// TIA Portal V20 export
DATA_BLOCK "DB_Components"   // DB119
// stored: InstanceOfName FB_Components, InstanceOfType FB
"FB_Components"
   // VAR
   //    sRT_Update : R_TRIG;
   //    sShuttle1DrilledPart : "FB_OPC_PartStatus";
   //    sShuttle1UndrilledPart { S7_SetPoint := 'True'} : "FB_OPC_PartStatus";
   //    sShuttle2DrilledPart { S7_SetPoint := 'True'} : "FB_OPC_PartStatus";
   //    sShuttle2UndrilledPart { S7_SetPoint := 'True'} : "FB_OPC_PartStatus";
   //    sShuttle1DrilledBw : "FB_OPC_PartStatus";
   //    sShuttle1UndrilledBw { S7_SetPoint := 'True'} : "FB_OPC_PartStatus";
   //    sShuttle2DrilledBw { S7_SetPoint := 'True'} : "FB_OPC_PartStatus";
   //    sShuttle2UndrilledBw { S7_SetPoint := 'True'} : "FB_OPC_PartStatus";
   //    sGripperDrilledPart : "FB_OPC_PartStatus";
   //    sGripperUndrilledPart { S7_SetPoint := 'True'} : "FB_OPC_PartStatus";
   //    sGripperDrilledBw : "FB_OPC_PartStatus";
   //    sGripperUndrilledBw { S7_SetPoint := 'True'} : "FB_OPC_PartStatus";
   //    sFixtureDrilledPart : "FB_OPC_PartStatus";
   //    sFixtureUndrilledPart { S7_SetPoint := 'True'} : "FB_OPC_PartStatus";
   //    sFixtureDrilledBw : "FB_OPC_PartStatus";
   //    sFixtureUndrilledBw { S7_SetPoint := 'True'} : "FB_OPC_PartStatus";
   // END_VAR
BEGIN
END_DATA_BLOCK
